FUNCTION_BLOCK geneticAlgorithmTest (* Event driven up counter *)
  (* Standard: 61499-1 Annex 2; Description: Copyright (c) 2017 fortiss GmbH This program and the accompanying materials are made available under the terms of the Eclipse Public License 2.0 which is available at https://www.eclipse.org/legal/epl-2.0/ SPDX-License-Identifier: EPL-2.0 *)
  (* Version 1.0, 2017-09-21, Alois Zoitl, fortiss GmbH, initial API and implementation and/or initial documentation *)
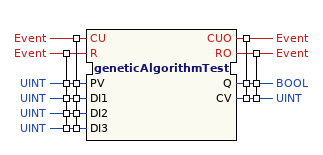
  EVENT_INPUT
    CU WITH PV, DI1, DI2, DI3; (* Count up *)
    R WITH PV, DI1, DI2, DI3; (* Reset *)
  END_EVENT
  EVENT_OUTPUT
    CUO WITH Q, CV; (* Count up output *)
    RO WITH Q, CV; (* Reset output *)
  END_EVENT
  VAR_INPUT
    PV : UINT := 0; (* Process Value *)
    DI1 : UINT := 0;
    DI2 : UINT := 0;
    DI3 : UINT := 0;
  END_VAR
  VAR_OUTPUT
    Q : BOOL := FALSE; (* True if CV &gt;= PV *)
    CV : UINT := 0; (* Counter Value *)
  END_VAR
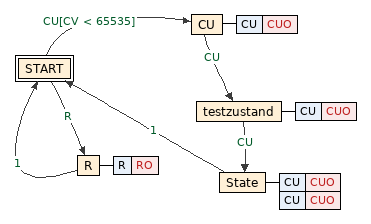
  EC_STATES
    START; (* Initial State *)
    CU : CU -> CUO;
    R : R -> RO;
    testzustand : CU -> CUO;
    State : CU -> CUO, CU -> CUO;
  END_STATES
  EC_TRANSITIONS
    START TO CU := CU[CV < 65535];
    START TO R := R;
    R TO START := 1;
    CU TO testzustand := CU;
    testzustand TO State := CU;
    State TO START := 1;
  END_TRANSITIONS
  ALGORITHM R IN ST:
CV := 0;
Q := FALSE;
  END_ALGORITHM
  ALGORITHM CU IN ST:
CV := CV + 1;
Q  := (CV >= PV);
  END_ALGORITHM
  SERVICE left interface/right interface (* Event driven up counter *)
    SEQUENCE Service Sequence
    END_SEQUENCE
    SEQUENCE Service Sequence
      left interface.R(PV:=0; DI1:=0; DI2:=0; DI3:=0;) -> left interface.RO();
      left interface.CU(PV:=0; DI1:=0; DI2:=0; DI3:=0;) -> left interface.CUO();
      left interface.R(PV:=0; DI1:=0; DI2:=0; DI3:=0;) -> left interface.RO();
      left interface.R(PV:=0; DI1:=0; DI2:=0; DI3:=0;) -> left interface.RO();
      left interface.CU(PV:=0; DI1:=0; DI2:=0; DI3:=0;) -> left interface.CUO();
      left interface.R(PV:=0; DI1:=0; DI2:=0; DI3:=0;) -> left interface.RO();
      left interface.R(PV:=0; DI1:=0; DI2:=0; DI3:=0;) -> left interface.RO();
      left interface.CU(PV:=0; DI1:=0; DI2:=0; DI3:=0;) -> left interface.CUO();
      left interface.CU(PV:=0; DI1:=0; DI2:=0; DI3:=0;) -> left interface.CUO();
      left interface.CU(PV:=0; DI1:=0; DI2:=0; DI3:=0;) -> left interface.CUO();
    END_SEQUENCE
  END_SERVICE
END_FUNCTION_BLOCK
